FUNCTION_BLOCK itfScaleAnalogInputImplement IMPLEMENTS itfScale
VAR_INPUT
END_VAR
VAR_OUTPUT
END_VAR
VAR
	AnalogSignal : INT;
	MaxSignalValue : INT;
	MaxUnitValue : INT;
	ScaledSignal : INT;
END_VAR

METHOD mScale : INT
pScaledSignal := pAnalogSignal * pMaxUnitValue / pMaxSignalValue;
END_METHOD

{warning 'add property implementation'}
PROPERTY pAnalogSignal : INT
GET
pAnalogSignal := AnalogSignal;
END_GET
SET
AnalogSignal := pAnalogSignal;
END_SET
END_PROPERTY

{warning 'add property implementation'}
PROPERTY pMaxSignalValue : INT
GET
IF MaxSignalValue > 0 THEN
pMaxSignalValue := MaxSignalValue;
ELSE
	pMaxSignalValue := 1;
END_IF
END_GET
SET
MaxSignalValue := pMaxSignalValue;
END_SET
END_PROPERTY

{warning 'add property implementation'}
PROPERTY pMaxUnitValue : INT
GET
pMaxUnitValue := MaxUnitValue;
END_GET
SET
MaxUnitValue := pMaxUnitValue;
END_SET
END_PROPERTY

{warning 'add property implementation'}
PROPERTY pScaledSignal : INT
GET
pScaledSignal := ScaledSignal;
END_GET
SET
ScaledSignal := pScaledSignal;
END_SET
END_PROPERTY

END_FUNCTION_BLOCK

(* stored: Version 1.1.0.1, ProductVersion 3.1.4024.12
   POU itfScaleAnalogInputImplement: Id {bd743808-21b2-4b7e-b273-88f12914b8a4}, SpecialFunc None
   Method mScale: Id {2cb0b6e4-b52c-44b2-9e28-fff038aec945}
   Property pAnalogSignal: Id {1045c361-c192-48cc-8fc0-a4af165b4924}
   Get Get: Id {1fe404f1-1b19-4cef-b5b1-afbe582d4781}
   Set Set: Id {ef2ddb16-9cd6-410a-8338-890e2e6f4414}
   Property pMaxSignalValue: Id {7ef7196e-d388-4ad4-9181-4e93c19fa8c0}
   Get Get: Id {6b0d6eb1-58d1-4202-aaff-92bba644abe9}
   Set Set: Id {06fd741b-1aed-408c-8e0c-25d7bbdde98e}
   Property pMaxUnitValue: Id {a2a01822-13f5-4f2b-84f3-5641ef38feff}
   Get Get: Id {ccdaca33-79e2-426c-8075-e8fea82ec24a}
   Set Set: Id {e6229e04-6729-46e3-ae36-6618bc1ef302}
   Property pScaledSignal: Id {d9a76f2c-a0f4-4965-be34-aca33c93e56a}
   Get Get: Id {eba4761e-cc4a-4433-a314-2da91daed415}
   Set Set: Id {e52c18d4-465d-4f88-ade3-2f828b8dd6cf} *)
